TYPE "Prod_Mode"
VERSION : 0.1
// Block: Prod_Mode
   STRUCT
      MES_ON : Bool;
      Cambio_Ordine_Automatico : Bool;
   END_STRUCT;

END_TYPE
